Universal Robots PolyScope program: Start Extrusion.urp

Program Start Extrusion (installation=default directory=/programs createdIn=5.14.5 lastSavedIn=5.21.3 robotSerialNumber=20246801938)
Calibrated DH parameters: a=[-0.000071, -0.790281, -0.600694, 0.000061, -0.000039, 0]; d=[0.236272, 604.465945, 132.116513, -736.382239, 0.159268, 0.154005]; alpha=[1.570254, -0.000567, 0.000559, 1.571709, -1.56999, 0]; deltaTheta=[0, -0.409357, 7.293326, -0.600784, -0.000001, -0.000001]
InitVariablesNode
Robot Program (runOnlyOnce=true)
  HwResp := "placeholder"
  SuppressedNode
    URCap WireTank Serial (WireTank Serial, WireTank, LLC) dataModel(Command=[252,72,49], NODE_TITLE=Serial Bridge uH1, byte_array=true, OUTPUT_ENTRY=Static, QUERY=false, Variable(key=OUTPUT_VARIABLE, variable=HwResp))
  ''
  ''
  Folder Folder1
    URCap WireTank Serial (WireTank Serial, WireTank, LLC) dataModel(NODE_TITLE=Serial Bridge uh?, Command=[252,104,63], byte_array=true, OUTPUT_ENTRY=Static, QUERY=true, Variable(key=OUTPUT_VARIABLE, variable(name=purge)))
    target := [252,72,49]
    resp := [1,2,3]
    URCap WireTank Serial (WireTank Serial, WireTank, LLC) dataModel(Command=[252,72,49], NODE_TITLE=Serial Bridge uH1, byte_array=true, QUERY=true, OUTPUT_ENTRY=Static, Variable(key=OUTPUT_VARIABLE, variable=resp))
    If resp≠target
      Popup Message (haltProgram=false message=could not confirm that heating started. check connection.  inputType=Text)
  SuppressedNode
    Wait Sleep waitTime=5
  SuppressedNode
    Popup Message (haltProgram=false message=heating started. push to stop inputType=Text)
  SuppressedNode
    URCap WireTank Serial (WireTank Serial, WireTank, LLC) dataModel(NODE_TITLE=Serial Bridge uh?, byte_array=true, Command=[252,104,63], OUTPUT_ENTRY=Static, QUERY=true, Variable(key=OUTPUT_VARIABLE, variable=HwResp))
  SuppressedNode
    Popup Message (haltProgram=false inputType=Variable) variable=HwResp
  SuppressedNode
    Wait Sleep waitTime=20
  SuppressedNode
    URCap WireTank Serial (WireTank Serial, WireTank, LLC) dataModel(byte_array=true, Command=[252,72,48], NODE_TITLE=Serial Bridge uH0, QUERY=false, OUTPUT_ENTRY=Static, Variable(key=OUTPUT_VARIABLE, variable=HwResp))
  SuppressedNode
    Popup Message (haltProgram=false message=heating stopped. push to start inputType=Text)
  'set the temp reader to high voltage (off) when program is running and low volt (on) when program not running'
  Script: set_runstate_standard_digital_output_to_value(2,3)
  'set 5V power to munsch powerbox to high (on) when a program is started and low on unscheduled stop'
  Script: set_runstate_standard_digital_output_to_value(1,5)
